# EPICS substitutions: ppmacApp/Db/autohome.substitutions
file "${PPMAC}/db/autohome.db"
{
pattern
{SYS,              DEV        PLC,  PORT  }
{"Prefix",  "Device",       0,    P0    }
}
